INTERFACE I_AxisDynamics EXTENDS I_Base

{attribute 'monitoring' := 'call'}
PROPERTY Acceleration : LREAL
GET
END_GET
SET
END_SET
END_PROPERTY

{attribute 'monitoring' := 'call'}
PROPERTY Deceleration : LREAL
GET
END_GET
SET
END_SET
END_PROPERTY

{attribute 'monitoring' := 'call'}
PROPERTY Jerk : LREAL
GET
END_GET
SET
END_SET
END_PROPERTY

{attribute 'monitoring' := 'call'}
PROPERTY Velocity : LREAL
GET
END_GET
SET
END_SET
END_PROPERTY

END_INTERFACE

(* stored: Version 1.1.0.1, ProductVersion 3.1.4026.20
   Itf I_AxisDynamics: Id {18131c95-6df6-45ac-9c87-9c2642fbb3bb}
   Property Acceleration: Id {f92ddbf9-7628-493c-b205-fa2781fafaf5}
   Get Get: Id {3d493785-b272-4d83-bd0b-0947c6c735b1}
   Set Set: Id {8ee4375b-d799-4d4c-9b2a-d7cfaf745448}
   Property Deceleration: Id {45bbf93d-209a-4ec7-9a59-a8ea3de9d573}
   Get Get: Id {d60516bb-39a3-4a89-97a0-2fd3c0dfff7a}
   Set Set: Id {15c19935-b1a4-4f47-bee7-c8d944e48399}
   Property Jerk: Id {ef83c49e-16f1-4ef8-ac47-0aad1d56be07}
   Get Get: Id {0327d9a1-d14a-49af-aabf-63701526741f}
   Set Set: Id {c2bfc0d3-60c5-4706-9027-f2f50f34021e}
   Property Velocity: Id {b7440370-a31f-4944-b6e3-353ff132589a}
   Get Get: Id {7cf26086-7e04-46f5-b179-40d32635c4d9}
   Set Set: Id {17aa3feb-a896-47c6-a417-e30f23acc1cf} *)
